Fanuc KAREL source: kc00025.KL

-- PROVISIONAL review KL for V940-1; original PC SHA256 7148c470831c3c9cd038e3ab50c899a894e30a7e9b243bf2fdce763503a37441
-- Incomplete behavior may be omitted. Consult companion uncertainty JSON. Do not deploy.
PROGRAM KC00025
%NOLOCKGROUP
BEGIN
  -- V9_ZERO_TABLE_METADATA_HINT layout=0002_ascii; no indexed target words; source/name/runtime held
  -- UNRESOLVED_PC offsets 5-17; opcodes 3F,75
  -- UNRESOLVED_PC offsets 22-64; opcodes 27,22,2A,22,22,22,22,22,31
  -- UNRESOLVED_PC offsets 69-73; opcodes 7F
END KC00025
